Fanuc KAREL source: kb00146.KL

-- PROVISIONAL review KL for V1013-1; original PC SHA256 c34442efdc85443b5440fb1c36c366aae60cf25d99b13db96ac36aab12102da0
-- Incomplete behavior may be omitted. Consult companion uncertainty JSON. Do not deploy.
PROGRAM KB00146
%NOLOCKGROUP
BEGIN
  -- UNRESOLVED_PC offsets 5-14; opcodes 3F,75
  -- UNRESOLVED_PC offsets 19-28; opcodes 3F,75
  -- UNRESOLVED_PC offsets 33-40; opcodes 9D,23
  -- UNRESOLVED_PC offsets 45-52; opcodes 9D,23
  -- UNRESOLVED_PC offsets 57-89; opcodes 27,22,2A,22,2A,22,22,31
  -- UNRESOLVED_PC offsets 94-98; opcodes 7F
END KB00146
